FUNCTION_BLOCK HHM_OV
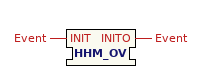
  EVENT_INPUT
    INIT;
  END_EVENT
  EVENT_OUTPUT
    INITO;
  END_EVENT
  FBS
    BEHAVIOUR : CMD_bloc;
    Trigger : ACTUORSbutton;
    ESTOP : EMGYSTOP;
    MODE : SELECT_MODE;
    STbutton : STARTandSTOP;
    ELcmd : AXE_CMD;
    ELplant : AXE_plant;
    CRcmd : AXE_CMD;
    CRplant : AXE_plant;
    CAcmd : AXE_CMD;
    CAplant : AXE_plant;
    GRplant : GR_plant;
    init : INITswitch;
    GRcmd : GR_CMD;
  END_FBS
  EVENT_CONNECTIONS
    ESTOP.INITO TO BEHAVIOUR.INIT;
    ELcmd.INITO TO ELplant.INIT;
    ELcmd.CNF TO ELplant.REQ;
    CRcmd.INITO TO CRplant.INIT;
    CRcmd.CNF TO CRplant.REQ;
    CRplant.CNF TO CRcmd.REQ;
    BEHAVIOUR.CNF TO ELcmd.REQ;
    BEHAVIOUR.CNF TO CRcmd.REQ;
    CAcmd.INITO TO CAplant.INIT;
    CAcmd.CNF TO CAplant.REQ;
    CAplant.CNF TO CAcmd.REQ;
    ELplant.CNF TO ELcmd.REQ;
    ELcmd.CNF TO BEHAVIOUR.REQ;
    CRcmd.CNF TO BEHAVIOUR.REQ;
    BEHAVIOUR.CNF TO CAcmd.REQ;
    CAcmd.CNF TO BEHAVIOUR.REQ;
    Trigger.INITO TO ESTOP.INIT;
    MODE.CNF TO BEHAVIOUR.REQ;
    STbutton.CNF TO BEHAVIOUR.REQ;
    ESTOP.CNF TO BEHAVIOUR.REQ;
    Trigger.CNF TO BEHAVIOUR.REQ;
    INIT TO STbutton.INIT;
    STbutton.INITO TO MODE.INIT;
    MODE.INITO TO init.INIT;
    init.INITO TO Trigger.INIT;
    init.CNF TO BEHAVIOUR.REQ;
    init.CNF TO CRcmd.REQ;
    init.CNF TO ELcmd.REQ;
    init.CNF TO CAcmd.REQ;
    CRcmd.CNF TO init.REQ;
    ELcmd.CNF TO init.REQ;
    CAcmd.CNF TO init.REQ;
    GRcmd.CNF TO GRplant.REQ;
    GRcmd.INITO TO GRplant.INIT;
    BEHAVIOUR.CNF TO GRcmd.REQ;
    BEHAVIOUR.INITO TO ELcmd.INIT;
    ELplant.INITO TO CRcmd.INIT;
    CRplant.INITO TO CAcmd.INIT;
    CAplant.INITO TO GRcmd.INIT;
    GRplant.INITO TO INITO;
    init.CNF TO GRcmd.REQ;
    GRcmd.CNF TO init.REQ;
    MODE.CNF TO Trigger.REQ;
    GRplant.CNF TO GRcmd.REQ;
  END_CONNECTIONS
  DATA_CONNECTIONS
    ESTOP.pressed TO BEHAVIOUR.ESTOP;
    STbutton.START TO BEHAVIOUR.START;
    STbutton.STOP TO BEHAVIOUR.STOP;
    Trigger.EL TO BEHAVIOUR.ELtriggered;
    Trigger.CR TO BEHAVIOUR.CRtriggered;
    Trigger.CA TO BEHAVIOUR.CAtriggered;
    Trigger.GR TO BEHAVIOUR.GRtriggered;
    ELcmd.go TO ELplant.GO;
    BEHAVIOUR.GOEL TO ELcmd.GO;
    BEHAVIOUR.SETEL TO ELcmd.SETPOS_IN;
    ELplant.PR TO ELcmd.PR;
    ELcmd.moving TO BEHAVIOUR.ELM;
    ELcmd.pr TO BEHAVIOUR.ELPR;
    CRcmd.go TO CRplant.GO;
    BEHAVIOUR.GOCR TO CRcmd.GO;
    BEHAVIOUR.SETCR TO CRcmd.SETPOS_IN;
    CRplant.PR TO CRcmd.PR;
    CRcmd.pr TO BEHAVIOUR.CRPR;
    CAcmd.go TO CAplant.GO;
    CAplant.PR TO CAcmd.PR;
    CAcmd.pr TO BEHAVIOUR.CAPR;
    BEHAVIOUR.GOCA TO CAcmd.GO;
    BEHAVIOUR.SETCA TO CAcmd.SETPOS_IN;
    MODE.MODE TO Trigger.MODE;
    init.SystemInited TO BEHAVIOUR.SystemINITED;
    GRcmd.open TO GRplant.OPEN;
    GRcmd.close TO GRplant.CLOSE;
    BEHAVIOUR.OPGR TO GRcmd.OPEN;
    BEHAVIOUR.CLGR TO GRcmd.CLOSE;
    GRplant.GRO TO GRcmd.openned;
    GRplant.GRC TO GRcmd.closed;
    GRcmd.GRO TO BEHAVIOUR.GRO;
    GRcmd.GRC TO BEHAVIOUR.GRC;
    CRcmd.moving TO BEHAVIOUR.CRM;
    CAcmd.moving TO BEHAVIOUR.CAM;
  END_CONNECTIONS
END_FUNCTION_BLOCK
